PROGRAM Auto_Cycle_Fix2
VAR
	Fixture_2 : Fix2_FB;
	TurnTable_1: TurnTable;
	Trunnion_1: Trunnion;
	RollerDoor_1: RollerDoor;
	Robot_Weld_1: Robot_Weld;
	Robot_MH_1: Robot_MH;
END_VAR
VAR // added by the converter: edge detectors and wires of the graphical bodies
    _w1, _w2 : BOOL;
END_VAR

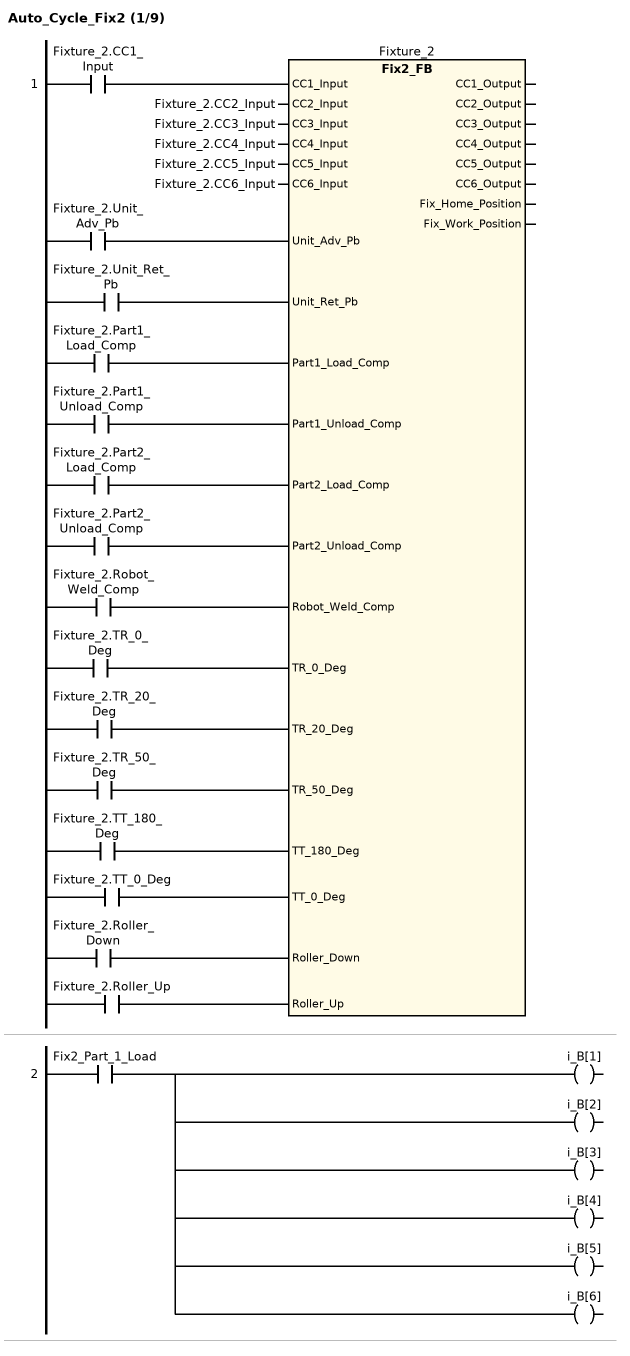
// NETWORK 1
Fixture_2(
    CC1_Input := Fixture_2.CC1_Input,
    CC2_Input := Fixture_2.CC2_Input,
    CC3_Input := Fixture_2.CC3_Input,
    CC4_Input := Fixture_2.CC4_Input,
    CC5_Input := Fixture_2.CC5_Input,
    CC6_Input := Fixture_2.CC6_Input,
    Unit_Adv_Pb := Fixture_2.Unit_Adv_Pb,
    Unit_Ret_Pb := Fixture_2.Unit_Ret_Pb,
    Part1_Load_Comp := Fixture_2.Part1_Load_Comp,
    Part1_Unload_Comp := Fixture_2.Part1_Unload_Comp,
    Part2_Load_Comp := Fixture_2.Part2_Load_Comp,
    Part2_Unload_Comp := Fixture_2.Part2_Unload_Comp,
    Robot_Weld_Comp := Fixture_2.Robot_Weld_Comp,
    TR_0_Deg := Fixture_2.TR_0_Deg,
    TR_20_Deg := Fixture_2.TR_20_Deg,
    TR_50_Deg := Fixture_2.TR_50_Deg,
    TT_180_Deg := Fixture_2.TT_180_Deg,
    TT_0_Deg := Fixture_2.TT_0_Deg,
    Roller_Down := Fixture_2.Roller_Down,
    Roller_Up := Fixture_2.Roller_Up); // Fix2_FB

// NETWORK 2
i_B[1] := Fix2_Part_1_Load;
i_B[2] := Fix2_Part_1_Load;
i_B[3] := Fix2_Part_1_Load;
i_B[4] := Fix2_Part_1_Load;
i_B[5] := Fix2_Part_1_Load;
i_B[6] := Fix2_Part_1_Load;

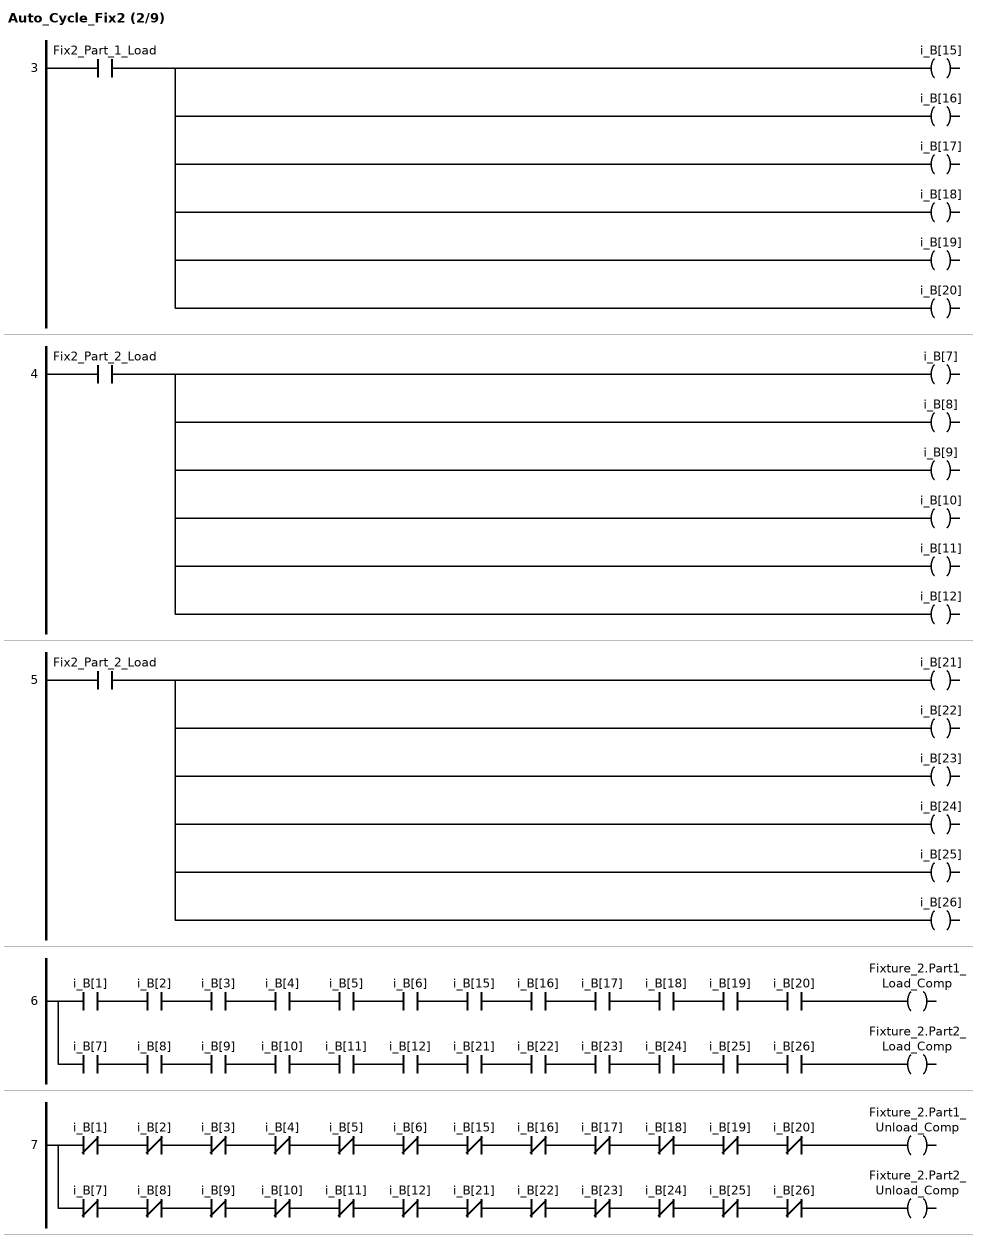
// NETWORK 3
i_B[15] := Fix2_Part_1_Load;
i_B[16] := Fix2_Part_1_Load;
i_B[17] := Fix2_Part_1_Load;
i_B[18] := Fix2_Part_1_Load;
i_B[19] := Fix2_Part_1_Load;
i_B[20] := Fix2_Part_1_Load;

// NETWORK 4
i_B[7] := Fix2_Part_2_Load;
i_B[8] := Fix2_Part_2_Load;
i_B[9] := Fix2_Part_2_Load;
i_B[10] := Fix2_Part_2_Load;
i_B[11] := Fix2_Part_2_Load;
i_B[12] := Fix2_Part_2_Load;

// NETWORK 5
i_B[21] := Fix2_Part_2_Load;
i_B[22] := Fix2_Part_2_Load;
i_B[23] := Fix2_Part_2_Load;
i_B[24] := Fix2_Part_2_Load;
i_B[25] := Fix2_Part_2_Load;
i_B[26] := Fix2_Part_2_Load;

// NETWORK 6
Fixture_2.Part1_Load_Comp := i_B[1] AND i_B[2] AND i_B[3] AND i_B[4] AND i_B[5] AND i_B[6] AND i_B[15] AND i_B[16] AND i_B[17] AND i_B[18] AND i_B[19] AND i_B[20];
Fixture_2.Part2_Load_Comp := i_B[7] AND i_B[8] AND i_B[9] AND i_B[10] AND i_B[11] AND i_B[12] AND i_B[21] AND i_B[22] AND i_B[23] AND i_B[24] AND i_B[25] AND i_B[26];

// NETWORK 7
Fixture_2.Part1_Unload_Comp := NOT i_B[1] AND NOT i_B[2] AND NOT i_B[3] AND NOT i_B[4] AND NOT i_B[5] AND NOT i_B[6] AND NOT i_B[15] AND NOT i_B[16] AND NOT i_B[17] AND NOT i_B[18] AND NOT i_B[19] AND NOT i_B[20];
Fixture_2.Part2_Unload_Comp := NOT i_B[7] AND NOT i_B[8] AND NOT i_B[9] AND NOT i_B[10] AND NOT i_B[11] AND NOT i_B[12] AND NOT i_B[21] AND NOT i_B[22] AND NOT i_B[23] AND NOT i_B[24] AND NOT i_B[25] AND NOT i_B[26];

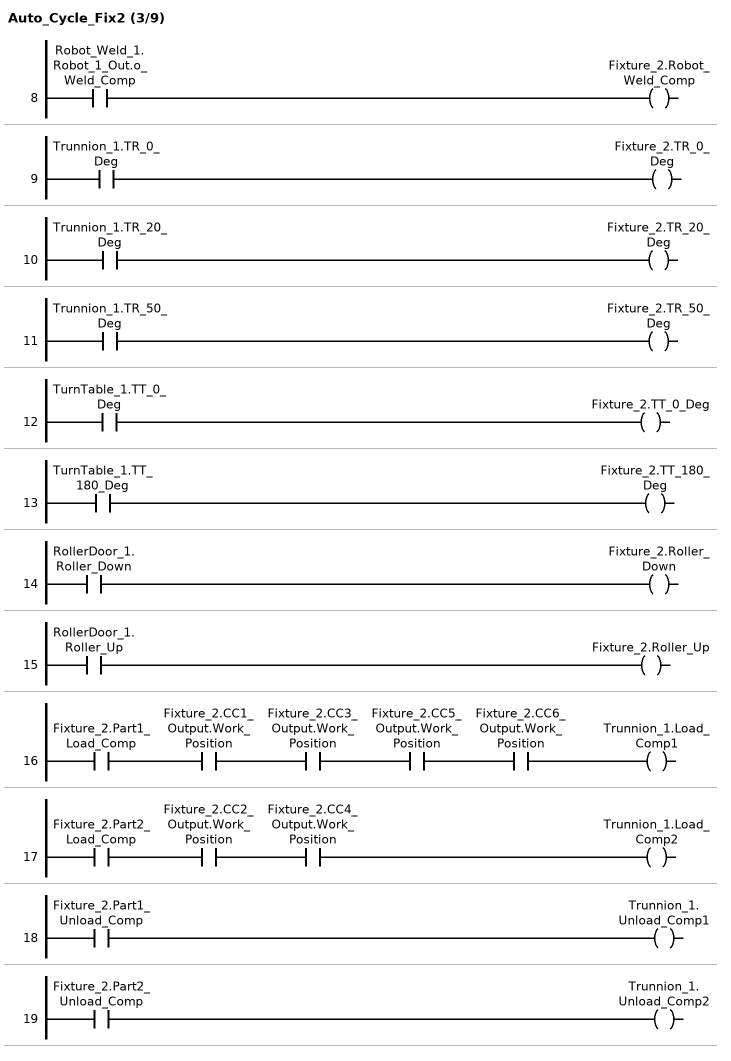
// NETWORK 8
Fixture_2.Robot_Weld_Comp := Robot_Weld_1.Robot_1_Out.o_Weld_Comp;

// NETWORK 9
Fixture_2.TR_0_Deg := Trunnion_1.TR_0_Deg;

// NETWORK 10
Fixture_2.TR_20_Deg := Trunnion_1.TR_20_Deg;

// NETWORK 11
Fixture_2.TR_50_Deg := Trunnion_1.TR_50_Deg;

// NETWORK 12
Fixture_2.TT_0_Deg := TurnTable_1.TT_0_Deg;

// NETWORK 13
Fixture_2.TT_180_Deg := TurnTable_1.TT_180_Deg;

// NETWORK 14
Fixture_2.Roller_Down := RollerDoor_1.Roller_Down;

// NETWORK 15
Fixture_2.Roller_Up := RollerDoor_1.Roller_Up;

// NETWORK 16
Trunnion_1.Load_Comp1 := Fixture_2.Part1_Load_Comp AND Fixture_2.CC1_Output.Work_Position AND Fixture_2.CC3_Output.Work_Position AND Fixture_2.CC5_Output.Work_Position AND Fixture_2.CC6_Output.Work_Position;

// NETWORK 17
Trunnion_1.Load_Comp2 := Fixture_2.Part2_Load_Comp AND Fixture_2.CC2_Output.Work_Position AND Fixture_2.CC4_Output.Work_Position;

// NETWORK 18
Trunnion_1.Unload_Comp1 := Fixture_2.Part1_Unload_Comp;

// NETWORK 19
Trunnion_1.Unload_Comp2 := Fixture_2.Part2_Unload_Comp;

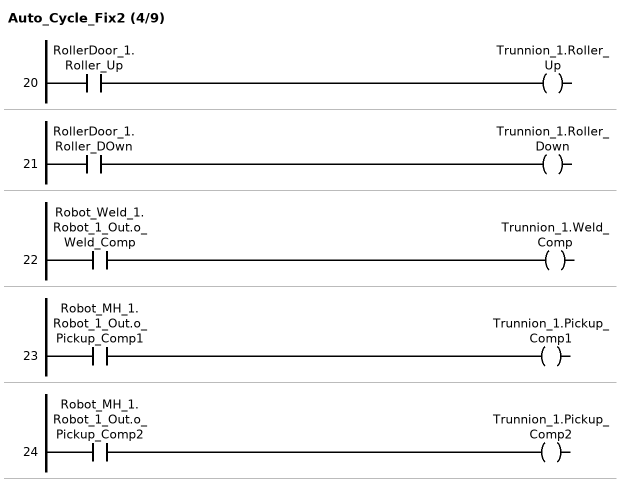
// NETWORK 20
Trunnion_1.Roller_Up := RollerDoor_1.Roller_Up;

// NETWORK 21
Trunnion_1.Roller_Down := RollerDoor_1.Roller_DOwn;

// NETWORK 22
Trunnion_1.Weld_Comp := Robot_Weld_1.Robot_1_Out.o_Weld_Comp;

// NETWORK 23
Trunnion_1.Pickup_Comp1 := Robot_MH_1.Robot_1_Out.o_Pickup_Comp1;

// NETWORK 24
Trunnion_1.Pickup_Comp2 := Robot_MH_1.Robot_1_Out.o_Pickup_Comp2;

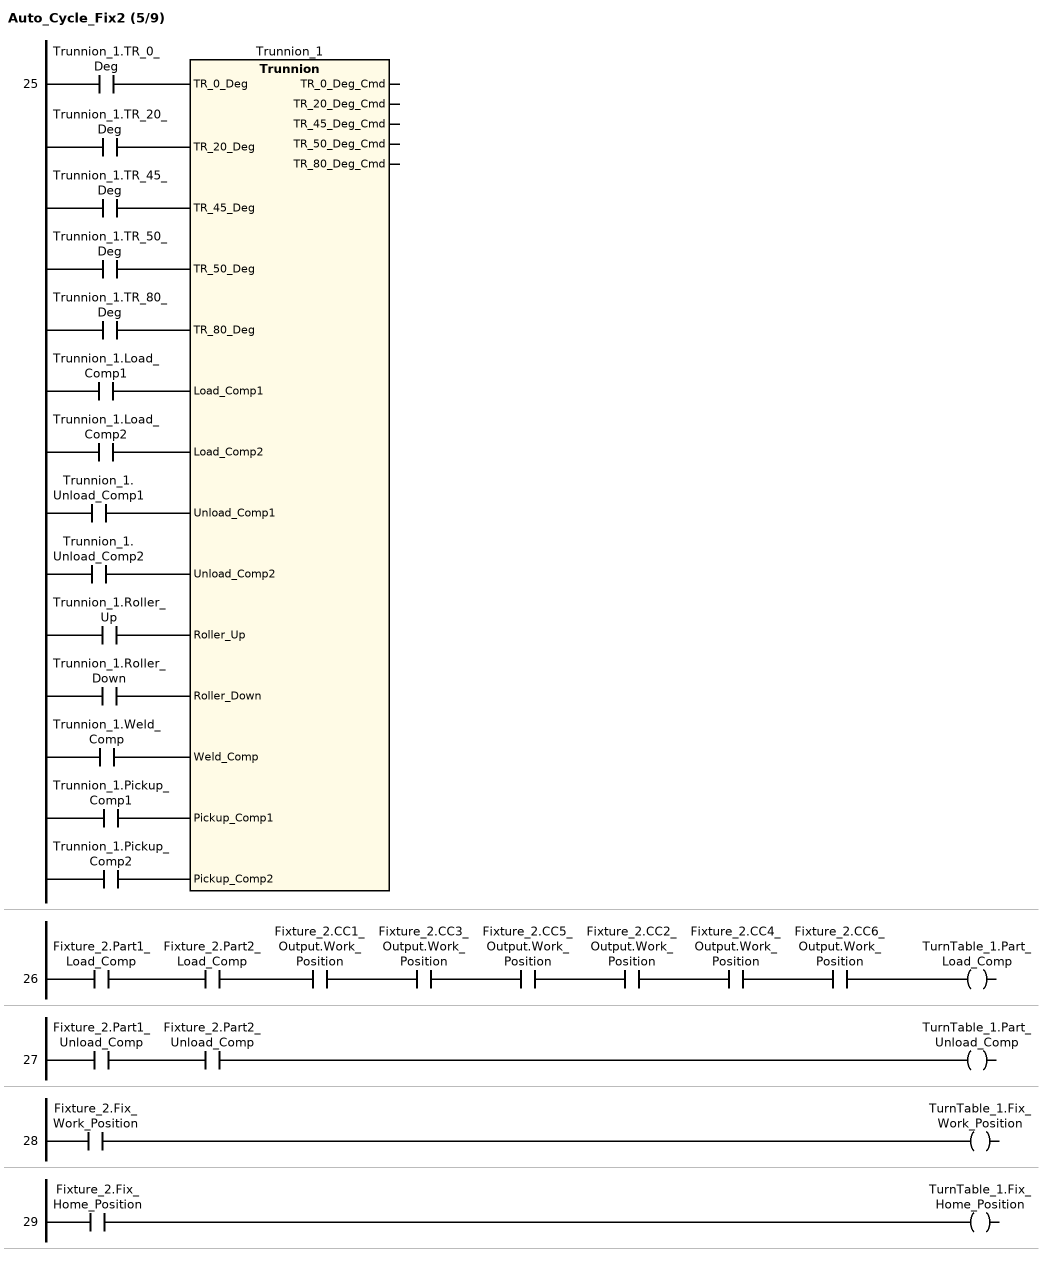
// NETWORK 25
Trunnion_1(
    TR_0_Deg := Trunnion_1.TR_0_Deg,
    TR_20_Deg := Trunnion_1.TR_20_Deg,
    TR_45_Deg := Trunnion_1.TR_45_Deg,
    TR_50_Deg := Trunnion_1.TR_50_Deg,
    TR_80_Deg := Trunnion_1.TR_80_Deg,
    Load_Comp1 := Trunnion_1.Load_Comp1,
    Load_Comp2 := Trunnion_1.Load_Comp2,
    Unload_Comp1 := Trunnion_1.Unload_Comp1,
    Unload_Comp2 := Trunnion_1.Unload_Comp2,
    Roller_Up := Trunnion_1.Roller_Up,
    Roller_Down := Trunnion_1.Roller_Down,
    Weld_Comp := Trunnion_1.Weld_Comp,
    Pickup_Comp1 := Trunnion_1.Pickup_Comp1,
    Pickup_Comp2 := Trunnion_1.Pickup_Comp2); // Trunnion

// NETWORK 26
TurnTable_1.Part_Load_Comp := Fixture_2.Part1_Load_Comp AND Fixture_2.Part2_Load_Comp AND Fixture_2.CC1_Output.Work_Position AND Fixture_2.CC3_Output.Work_Position AND Fixture_2.CC5_Output.Work_Position AND Fixture_2.CC2_Output.Work_Position AND Fixture_2.CC4_Output.Work_Position AND Fixture_2.CC6_Output.Work_Position;

// NETWORK 27
TurnTable_1.Part_Unload_Comp := Fixture_2.Part1_Unload_Comp AND Fixture_2.Part2_Unload_Comp;

// NETWORK 28
TurnTable_1.Fix_Work_Position := Fixture_2.Fix_Work_Position;

// NETWORK 29
TurnTable_1.Fix_Home_Position := Fixture_2.Fix_Home_Position;

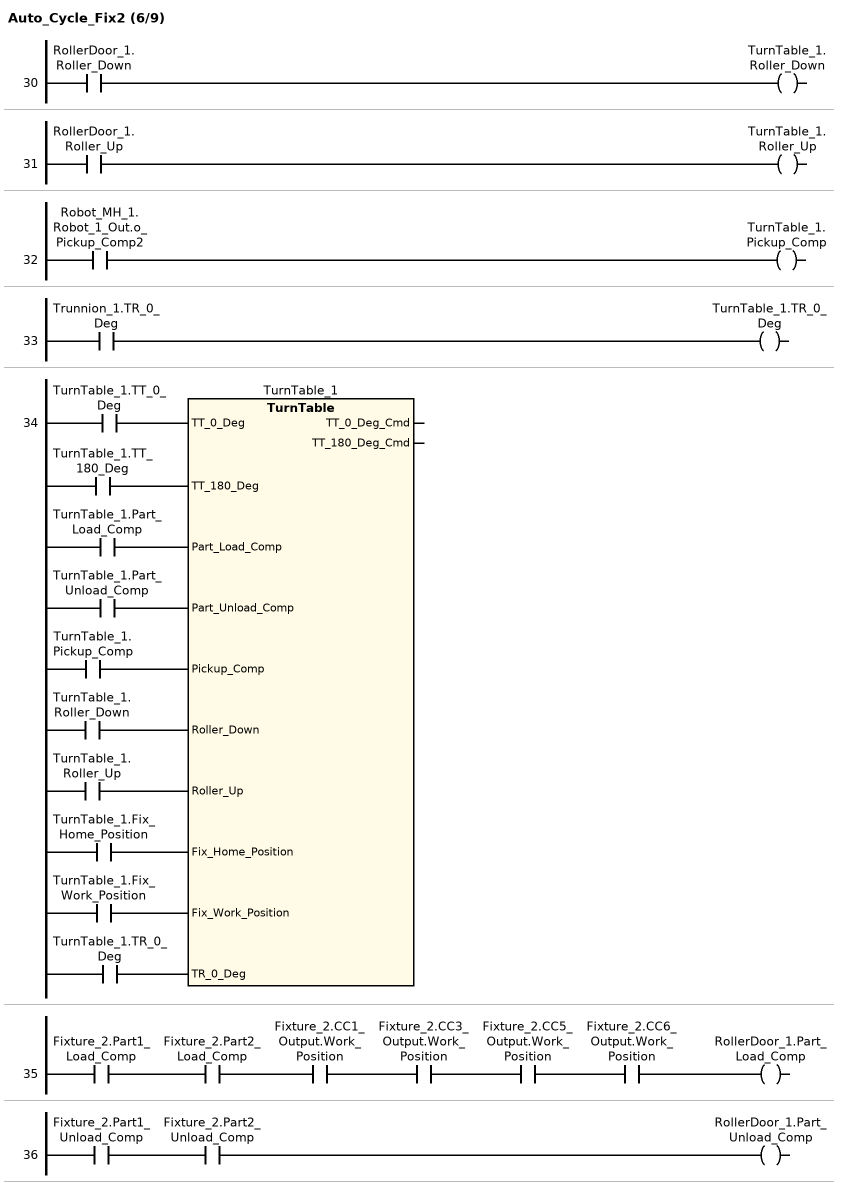
// NETWORK 30
TurnTable_1.Roller_Down := RollerDoor_1.Roller_Down;

// NETWORK 31
TurnTable_1.Roller_Up := RollerDoor_1.Roller_Up;

// NETWORK 32
TurnTable_1.Pickup_Comp := Robot_MH_1.Robot_1_Out.o_Pickup_Comp2;

// NETWORK 33
TurnTable_1.TR_0_Deg := Trunnion_1.TR_0_Deg;

// NETWORK 34
TurnTable_1(
    TT_0_Deg := TurnTable_1.TT_0_Deg,
    TT_180_Deg := TurnTable_1.TT_180_Deg,
    Part_Load_Comp := TurnTable_1.Part_Load_Comp,
    Part_Unload_Comp := TurnTable_1.Part_Unload_Comp,
    Pickup_Comp := TurnTable_1.Pickup_Comp,
    Roller_Down := TurnTable_1.Roller_Down,
    Roller_Up := TurnTable_1.Roller_Up,
    Fix_Home_Position := TurnTable_1.Fix_Home_Position,
    Fix_Work_Position := TurnTable_1.Fix_Work_Position,
    TR_0_Deg := TurnTable_1.TR_0_Deg); // TurnTable

// NETWORK 35
RollerDoor_1.Part_Load_Comp := Fixture_2.Part1_Load_Comp AND Fixture_2.Part2_Load_Comp AND Fixture_2.CC1_Output.Work_Position AND Fixture_2.CC3_Output.Work_Position AND Fixture_2.CC5_Output.Work_Position AND Fixture_2.CC6_Output.Work_Position;

// NETWORK 36
RollerDoor_1.Part_Unload_Comp := Fixture_2.Part1_Unload_Comp AND Fixture_2.Part2_Unload_Comp;

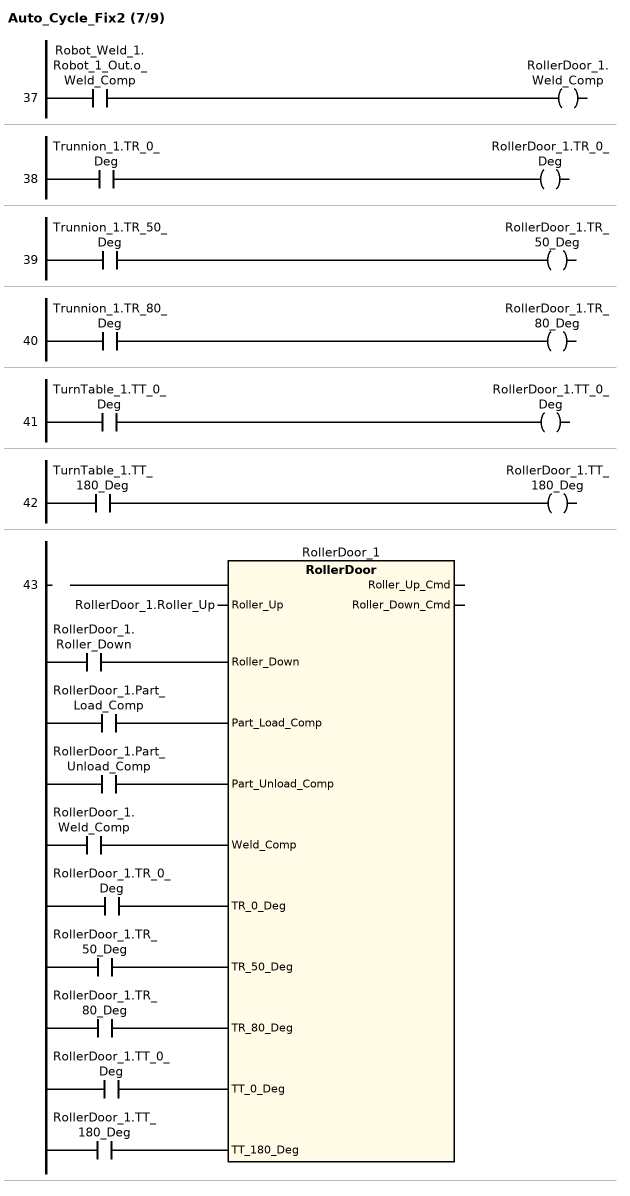
// NETWORK 37
RollerDoor_1.Weld_Comp := Robot_Weld_1.Robot_1_Out.o_Weld_Comp;

// NETWORK 38
RollerDoor_1.TR_0_Deg := Trunnion_1.TR_0_Deg;

// NETWORK 39
RollerDoor_1.TR_50_Deg := Trunnion_1.TR_50_Deg;

// NETWORK 40
RollerDoor_1.TR_80_Deg := Trunnion_1.TR_80_Deg;

// NETWORK 41
RollerDoor_1.TT_0_Deg := TurnTable_1.TT_0_Deg;

// NETWORK 42
RollerDoor_1.TT_180_Deg := TurnTable_1.TT_180_Deg;

// NETWORK 43
RollerDoor_1(
    Roller_Up := RollerDoor_1.Roller_Up,
    Roller_Down := RollerDoor_1.Roller_Down,
    Part_Load_Comp := RollerDoor_1.Part_Load_Comp,
    Part_Unload_Comp := RollerDoor_1.Part_Unload_Comp,
    Weld_Comp := RollerDoor_1.Weld_Comp,
    TR_0_Deg := RollerDoor_1.TR_0_Deg,
    TR_50_Deg := RollerDoor_1.TR_50_Deg,
    TR_80_Deg := RollerDoor_1.TR_80_Deg,
    TT_0_Deg := RollerDoor_1.TT_0_Deg,
    TT_180_Deg := RollerDoor_1.TT_180_Deg); // RollerDoor

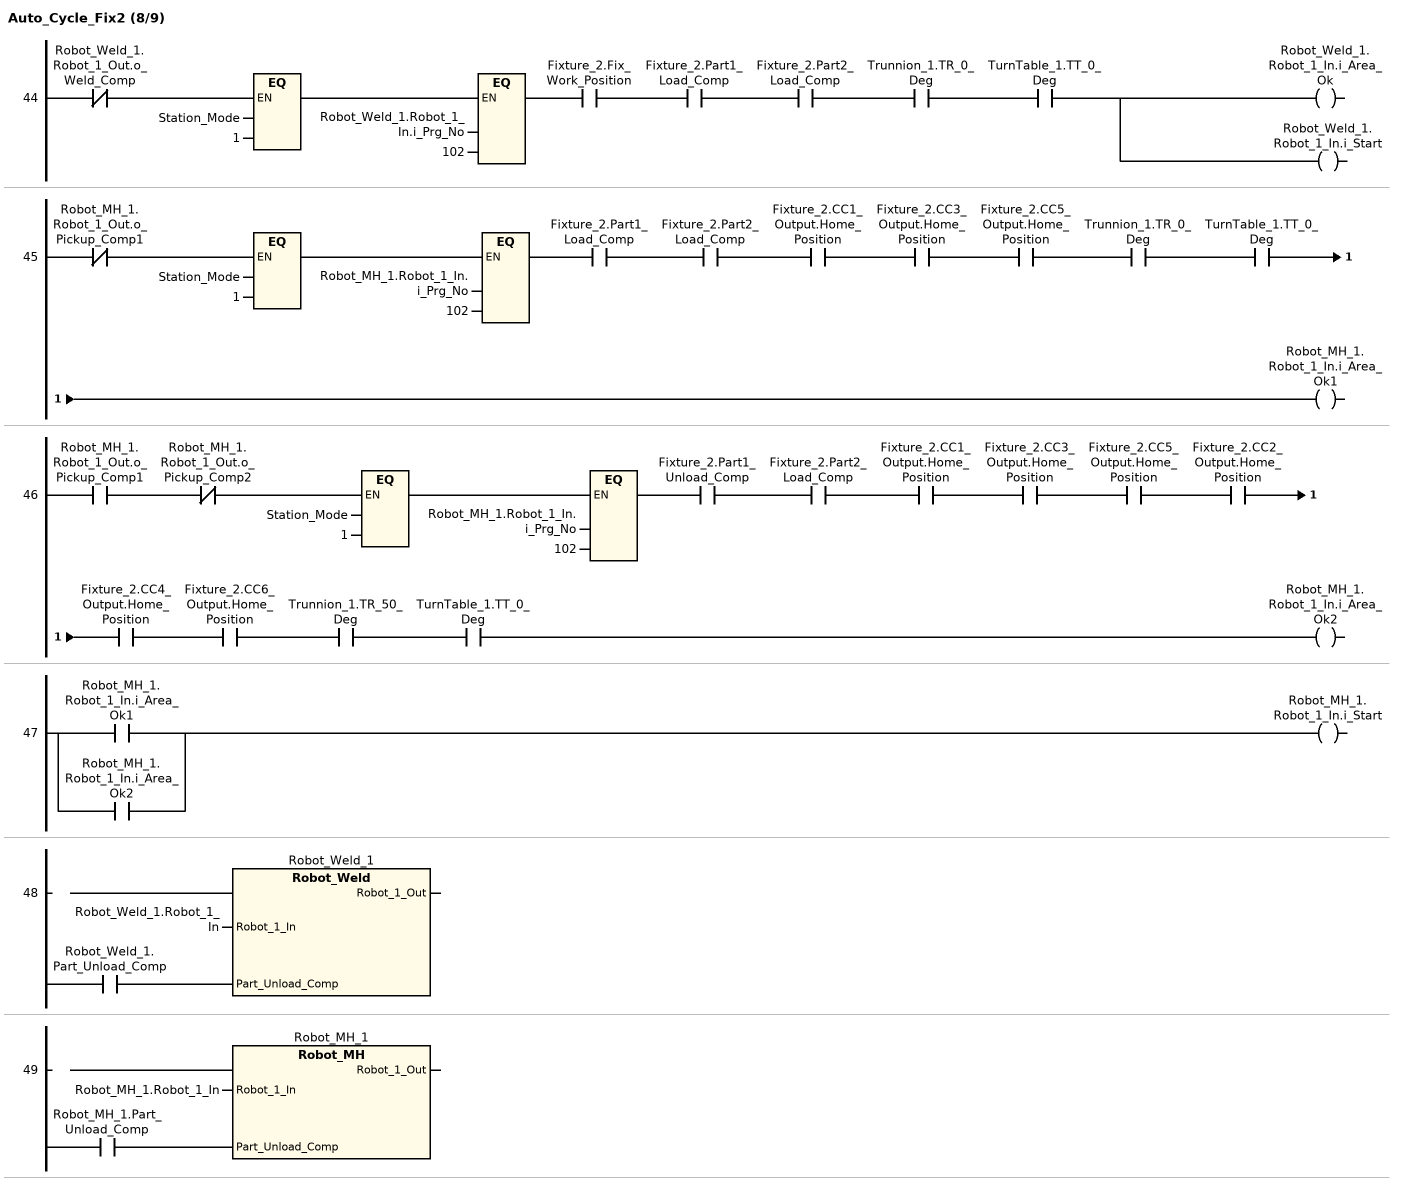
// NETWORK 44
_w1 := (NOT Robot_Weld_1.Robot_1_Out.o_Weld_Comp AND Station_Mode = 1 AND Robot_Weld_1.Robot_1_In.i_Prg_No = 102) AND Fixture_2.Fix_Work_Position AND Fixture_2.Part1_Load_Comp AND Fixture_2.Part2_Load_Comp AND Trunnion_1.TR_0_Deg AND TurnTable_1.TT_0_Deg;
Robot_Weld_1.Robot_1_In.i_Area_Ok := _w1;
Robot_Weld_1.Robot_1_In.i_Start := _w1;

// NETWORK 45
Robot_MH_1.Robot_1_In.i_Area_Ok1 := (NOT Robot_MH_1.Robot_1_Out.o_Pickup_Comp1 AND Station_Mode = 1 AND Robot_MH_1.Robot_1_In.i_Prg_No = 102) AND Fixture_2.Part1_Load_Comp AND Fixture_2.Part2_Load_Comp AND Fixture_2.CC1_Output.Home_Position AND Fixture_2.CC3_Output.Home_Position AND Fixture_2.CC5_Output.Home_Position AND Trunnion_1.TR_0_Deg AND TurnTable_1.TT_0_Deg;

// NETWORK 46
Robot_MH_1.Robot_1_In.i_Area_Ok2 := (Robot_MH_1.Robot_1_Out.o_Pickup_Comp1 AND NOT Robot_MH_1.Robot_1_Out.o_Pickup_Comp2 AND Station_Mode = 1 AND Robot_MH_1.Robot_1_In.i_Prg_No = 102) AND Fixture_2.Part1_Unload_Comp AND Fixture_2.Part2_Load_Comp AND Fixture_2.CC1_Output.Home_Position AND Fixture_2.CC3_Output.Home_Position AND Fixture_2.CC5_Output.Home_Position AND Fixture_2.CC2_Output.Home_Position AND Fixture_2.CC4_Output.Home_Position AND Fixture_2.CC6_Output.Home_Position AND Trunnion_1.TR_50_Deg AND TurnTable_1.TT_0_Deg;

// NETWORK 47
Robot_MH_1.Robot_1_In.i_Start := Robot_MH_1.Robot_1_In.i_Area_Ok1 OR Robot_MH_1.Robot_1_In.i_Area_Ok2;

// NETWORK 48
Robot_Weld_1(Robot_1_In := Robot_Weld_1.Robot_1_In, Part_Unload_Comp := Robot_Weld_1.Part_Unload_Comp); // Robot_Weld

// NETWORK 49
Robot_MH_1(Robot_1_In := Robot_MH_1.Robot_1_In, Part_Unload_Comp := Robot_MH_1.Part_Unload_Comp); // Robot_MH

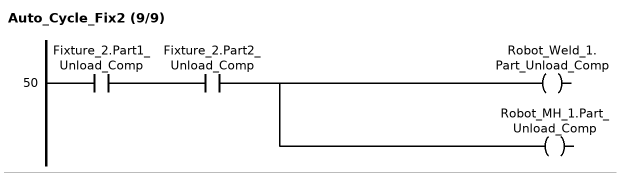
// NETWORK 50
_w2 := Fixture_2.Part1_Unload_Comp AND Fixture_2.Part2_Unload_Comp;
Robot_Weld_1.Part_Unload_Comp := _w2;
Robot_MH_1.Part_Unload_Comp := _w2;

END_PROGRAM

(* stored: Version 1.1.0.1, ProductVersion 3.1.4024.16
   POU Auto_Cycle_Fix2: Id {b45f7483-7299-4d7b-8624-4a90ce87e627}, SpecialFunc None *)
